{attribute 'qualified_only'}
{attribute 'strict'}
TYPE E_Test_NotificationId :
(
	OnPbPressed_Notification := 1000,
    
    MaxNotificationId
) UDINT;
END_TYPE

(* stored: Version 1.1.0.1, ProductVersion 3.1.4024.5
   DUT E_Test_NotificationId: Id {29196a41-8736-4c5c-99db-9777ba708e06} *)
